INTERFACE I_Event

PROPERTY Name : T_MaxString
GET
END_GET
END_PROPERTY

END_INTERFACE

(* stored: Version 1.1.0.1, ProductVersion 3.1.4024.12
   Itf I_Event: Id {ea7febc2-8479-4f67-a091-10e07f511835}
   Property Name: Id {9368da16-cdb5-4c27-8620-fdba96a21a0b}
   Get Get: Id {edc8f2e5-c147-46b0-84bf-3adc39448d47} *)
